INTERFACE ITF_TopElement2 EXTENDS ITF_BaseTopElement

END_INTERFACE

(* stored: Version 1.1.0.1, ProductVersion 3.1.4024.15
   Itf ITF_TopElement2: Id {0cbde385-5cf5-427e-87cb-b340151cc3ce} *)
